(* PLC project PLC107_AI, home PLC107_AI 1 *)
(* stored: creationDateTime 2019-11-13T09:37:45, productRelease 0, modificationDateTime 2020-07-16T10:33:36, version 1 *)

(* Установка режима работы аналогового входа *)
FUNCTION_BLOCK AIMode
  VAR_INPUT
    Ex : BOOL := FALSE;  (* разрешение на выполнение *)
    AIn : BYTE := 0;  (* номер входа *)
    M : BYTE := 0;  (* режим работы *)
  END_VAR
  VAR_OUTPUT
    Om : BYTE := 0;  (* режим работы (установленный) *)
    Os : BYTE := 0;  (* код состояния входа *)
    Ok : BYTE := 0;  (* код результата исполнения блока *)
  END_VAR

            {extern void App_AIMode(AIMODE*);App_AIMode(data__);}

          
END_FUNCTION_BLOCK

(* Получение значения аналогового входа *)
FUNCTION_BLOCK AIVal
  VAR_INPUT
    Ex : BOOL := FALSE;  (* разрешение на выполнение *)
    AIn : BYTE := 0;  (* номер входа *)
  END_VAR
  VAR_OUTPUT
    Ov : REAL := 0.0;  (* значение *)
    Os : BYTE := 0;  (* код состояния *)
    Ok : BYTE := 0;  (* код результата исполнения блока *)
  END_VAR

            {extern void App_AIVal(AIVAL*);App_AIVal(data__);}

          
END_FUNCTION_BLOCK
